FUNCTION_BLOCK JoinAllClosestTracks IMPLEMENTS I_DemoStep, I_XplanarTable
VAR_INPUT
	XPlanarSys		: 	I_XPlanarSystem;
	UseOrientation : BOOL := FALSE;
END_VAR
VAR_OUTPUT
END_VAR
VAR
	_Done				: BOOL;
END_VAR

METHOD CyclicLogic
//E_DemoStep.JoinTrack:
IF XPlanarSys.EnableTracks().Done AND 
	ip.Movers[1].MoveCommand.JoinClosestTrack(UseOrientation).Done AND
	ip.Movers[2].MoveCommand.JoinClosestTrack(UseOrientation).Done 
THEN
	_Done:=TRUE;
END_IF
END_METHOD

{attribute 'monitoring' := 'call'}
PROPERTY Done : BOOL
GET
Done:= _Done;
END_GET
END_PROPERTY

METHOD Reset : BOOL
_Done:=FALSE;
Reset:=TRUE;
END_METHOD

PROPERTY Table : I_XPlanarSystem
GET
Table:=XPlanarSys;
END_GET
SET
XPlanarSys:=Table;
END_SET
END_PROPERTY

END_FUNCTION_BLOCK

(* stored: Version 1.1.0.1, ProductVersion 3.1.4026.20
   POU JoinAllClosestTracks: Id {42b93498-6f63-4169-82ce-f7c0f205be7d}, SpecialFunc None
   Method CyclicLogic: Id {f02fb9b8-f251-4a83-bdbe-877fedfb106d}
   Property Done: Id {3e1a5e81-419b-4c2a-8221-60dcf82fdbb7}
   Get Get: Id {ea12fd83-43ae-4d12-bcb8-2870791efc64}
   Method Reset: Id {75077b62-9d74-49d1-bc7a-01692252d5f7}
   Property Table: Id {5cb14338-6d41-4365-b5b3-a7d0ef616e3a}
   Get Get: Id {af8818ea-2f47-4007-b873-73532957033e}
   Set Set: Id {02051645-4c0f-4f68-8c7f-6ebf7a9ebcae} *)
